Yaskawa INFORM job: CM_PRINT.JBI

/JOB
//NAME CM_PRINT
//POS
///NPOS 0,0,0,0,0,0
//INST
///DATE 2025/02/20 16:20
///COMM Generated using RoboDK
///ATTR SC,RW
///GROUP1 RB1
NOP
CALL JOB:PRINT3D
CALL JOB:PRINT3D2
CALL JOB:PRINT3D3
CALL JOB:PRINT3D4
CALL JOB:PRINT3D5
CALL JOB:PRINT3D6
CALL JOB:PRINT3D7
CALL JOB:PRINT3D8
CALL JOB:PRINT3D9
CALL JOB:PRINT3D10
CALL JOB:PRINT3D11
CALL JOB:PRINT3D12
CALL JOB:PRINT3D13
CALL JOB:PRINT3D14
CALL JOB:PRINT3D15
CALL JOB:PRINT3D16
CALL JOB:PRINT3D17
CALL JOB:PRINT3D18
END
